TYPE ST_PowerGroupParCmd :
STRUCT
    SchemaVersion : UINT := 1;
END_STRUCT
END_TYPE

(* stored: Version 1.1.0.1, ProductVersion 3.1.4024.12
   DUT ST_PowerGroupParCmd: Id {212915f6-ae88-45d4-a659-184f1952254f} *)
